{attribute 'qualified_only'}
VAR_GLOBAL CONSTANT 
	//debug
	uiHistoStep_C								        : INT := 50;
END_VAR

(* stored: Version 1.1.0.1, ProductVersion 3.1.4024.12
   GVL C: Id {f2d0c7e9-6162-4f20-8df8-b91ac86dab85} *)
